// TIA Portal V19 export
VAR_GLOBAL   // PLC tag table "Default tag table"
   "AN IN 1" AT %IW113 : Int;
   "AN IN 2" AT %IW115 : Int;
   "AN IN 3" AT %IW117 : Int;
   "AN IN 4" AT %IW119 : Int;
   "DI 0.0" AT %I0.0 : Bool;
   "DI 0.1" AT %I0.1 : Bool;
   "DI 0.2" AT %I0.2 : Bool;
   "DI 0.3" AT %I0.3 : Bool;
   "DI 0.4" AT %I0.4 : Bool;
   "DI 0.5" AT %I0.5 : Bool;
   "DI 0.6" AT %I0.6 : Bool;
   "DI 0.7" AT %I0.7 : Bool;
   "DI 1.0" AT %I1.0 : Bool;
   "DI 1.1" AT %I1.1 : Bool;
   "DI 1.2" AT %I1.2 : Bool;
   "DI 1.3" AT %I1.3 : Bool;
   "DI 1.4" AT %I1.4 : Bool;
   "DI 1.5" AT %I1.5 : Bool;
   FmMassFlow AT %ID68 : Real;
   "FmVolume Flow" AT %ID73 : Real;
   FmMassFlow_Sts AT %IB72 : Byte;
   "FmVolume Flow_Sts" AT %IB77 : Byte;
   FmCorrectedVolumeFlow AT %ID78 : Real;
   FmCorrectedVolumeFlowSts AT %IB82 : Byte;
   FMDensity AT %ID83 : Real;
   FMDensitySts AT %IB87 : Byte;
   FmReferenceDensity AT %ID88 : Real;
   FMReferenceDensitySts AT %IB92 : Byte;
   FmTemperature AT %ID93 : Real;
   FMTemperatureSts AT %IB97 : Byte;
   FMTotalizer1Read AT %ID98 : Real;
   FMTotaliser1Sts AT %IB102 : Byte;
   "DQ 0.0" AT %Q0.0 : Bool;
   "DQ 0.1" AT %Q0.1 : Bool;
   "DQ 0.2" AT %Q0.2 : Bool;
   "DQ 0.3" AT %Q0.3 : Bool;
   "DQ 0.4" AT %Q0.4 : Bool;
   "DQ 0.5" AT %Q0.5 : Bool;
   "DQ 0.6" AT %Q0.6 : Bool;
   "DQ 0.7" AT %Q0.7 : Bool;
   "DQ 1.0" AT %Q1.0 : Bool;
   "DQ 1.1" AT %Q1.1 : Bool;
   FMTotaliser1Control AT %QB64 : Byte;
   System_Byte AT %MB1 : Byte;
   FirstScan AT %M1.0 : Bool;
   DiagStatusUpdate AT %M1.1 : Bool;
   AlwaysTRUE AT %M1.2 : Bool;
   AlwaysFALSE AT %M1.3 : Bool;
   Clock_Byte AT %MB0 : Byte;
   Clock_10Hz AT %M0.0 : Bool;
   Clock_5Hz AT %M0.1 : Bool;
   "Clock_2.5Hz" AT %M0.2 : Bool;
   Clock_2Hz AT %M0.3 : Bool;
   "Clock_1.25Hz" AT %M0.4 : Bool;
   Clock_1Hz AT %M0.5 : Bool;
   "Clock_0.625Hz" AT %M0.6 : Bool;
   "Clock_0.5Hz" AT %M0.7 : Bool;
   "Request Run Motor Cooling" AT %M2.0 : Bool;
   StopPump AT %M2.1 : Bool;
   VFDCmdRun AT %M2.2 : Bool;
   CMDDose AT %M2.3 : Bool;
   OpenFlowmeterValve AT %M2.4 : Bool;
   OpenDoseValve AT %M2.5 : Bool;
   StopDoseVal AT %M2.6 : Bool;
   RepeatDose AT %M2.7 : Bool;
   StopDoseTime AT %M3.0 : Bool;
   LatchRPTStart AT %M3.1 : Bool;
   LatchRPTStop AT %M3.2 : Bool;
   FaultReset AT %M3.3 : Bool;
   Simulation AT %M3.4 : Bool;
   DoseVLVOpnFLT AT %M3.5 : Bool;
   DoseVLVClsFLT AT %M3.6 : Bool;
   OpenIBCValve AT %M3.7 : Bool;
   OpenPumpValve AT %M4.0 : Bool;
   IBCVLVOpnFLT AT %M4.1 : Bool;
   IBCVLVClsFLT AT %M4.2 : Bool;
   PumpVLVOpnFLT AT %M4.3 : Bool;
   PumpVLVClsFLT AT %M4.4 : Bool;
   FlVLVOpnFLT AT %M4.5 : Bool;
   FlVLVClsFLT AT %M4.6 : Bool;
   TestFmVals AT %MD6 : Real;
   trigStore1 AT %M4.7 : Bool;
   AlarmStoreCount AT %MD10 : Real;
   StopSystemNoDOse AT %M5.0 : Bool;
   AlarmLookForNoChange AT %M5.1 : Bool;
   "HMI Start TImer" AT %M5.2 : Bool;
   "HMI Timer Set Value" AT %MD14 : Time;
   "HMI timer alarm" AT %M18.0 : Bool;
   "time write sts" AT %MW1142 : Int;
   "time  read sts" AT %MW1168 : Int;
   "Time Write" AT %M148.4 : Bool;
   alarmTAG1 AT %MW148 : Int;
   Simulate AT %M5.3 : Bool;
   PumpIsRunning AT %M5.4 : Bool;
   sim_flow AT %MD20 : Real;
END_VAR
